FUNCTION_BLOCK Farbe (* Basic Function Block Type *)
  (* Standard: 61499-2 *)
  (* Version 0.0, 21/06/2022, Lernfabrik, WBK hackaton, Template *)
  PACKAGE Main;
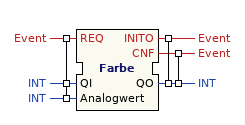
  EVENT_INPUT
    REQ WITH QI, Analogwert; (* Normal Execution Request *)
  END_EVENT
  EVENT_OUTPUT
    INITO WITH QO; (* Initialization Confirm *)
    CNF WITH QO; (* Execution Confirmation *)
  END_EVENT
  VAR_INPUT
    QI : INT; (* Input event qualifier *)
    Analogwert : INT;
  END_VAR
  VAR_OUTPUT
    QO : INT; (* Output event qualifier *)
  END_VAR
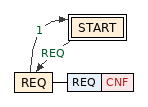
  EC_STATES
    START; (* Initial State *)
    REQ : REQ -> CNF; (* Normal execution *)
  END_STATES
  EC_TRANSITIONS
    START TO REQ := REQ;
    REQ TO START := 1;
  END_TRANSITIONS
  ALGORITHM INIT IN ST: (* Initialization algorithm *)
;
  END_ALGORITHM
  ALGORITHM REQ IN ST: (* Normally executed algorithm *)
QO := QI / Analogwert;
;
  END_ALGORITHM
END_FUNCTION_BLOCK
